TYPE SafetyEmergencyStopsStatuses :
STRUCT
	///Are the emergency stops in a healthy state? Good=RUN, Bad=safe stopped
	healthStatus: HealthStatus;
	///Is the safety busy?
	busyStatus: BusyStatus;
END_STRUCT
END_TYPE

(* stored: Version 1.1.0.1, ProductVersion 3.1.4019.2
   DUT SafetyEmergencyStopsStatuses: Id {e4809a7c-6ce7-4533-b00a-10fd747e96d8} *)
